FUNCTION TryConvert_SINT_TO_LREAL : BOOL
VAR_INPUT
	in : SINT;
	out : REFERENCE TO LREAL;
END_VAR

out := SINT_TO_LREAL(in);
TryConvert_SINT_TO_LREAL := TRUE;

END_FUNCTION

(* stored: Version 1.1.0.1, ProductVersion 3.1.4024.12
   POU TryConvert_SINT_TO_LREAL: Id {481e0bd5-9aef-4779-a3f2-9eff0a567c4c}, SpecialFunc None *)
